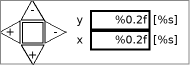
VISUALIZATION _VISU_PlacementXY_cross  // 190x65
VAR_IN_OUT
	m_Inst : FB_PointCorr;  
END_VAR
    Polyline (21,20) (32,0) (44,20) (21,20), "-"
        p3092690914: m_Inst.nBtnColor
        tap m_Inst.bCmd_Y_minus
    Polyline (21,45) (33,65) (44,45) (21,45), "+"
        p3092690914: m_Inst.nBtnColor
        tap m_Inst.bCmd_Y_plus
    Polyline (45,43) (45,21) (66,32) (45,43), "-"
        p3092690914: m_Inst.nBtnColor
        tap m_Inst.bCmd_X_minus
    Polyline (20,43) (20,21) (0,32) (20,43), "+"
        p3092690914: m_Inst.nBtnColor
        tap m_Inst.bCmd_X_plus
    Rectangle (70,30 20x20), "x"
    Rectangle (70,10 20x20), "y"
    Rectangle (22,22 21x21)
    Rectangle (150,10 40x20), "[%s]", text variable: m_Inst._aUnit
    Rectangle (150,30 40x20), "[%s]", text variable: m_Inst._aUnit
    Rectangle (90,10 60x20), "%0.2f", text variable: m_Inst.fY_Pos
        OnMouseClick: write the text variable via Default
    Rectangle (90,30 60x20), "%0.2f", text variable: m_Inst.fX_Pos
        OnMouseClick: write the text variable via Default
END_VISUALIZATION

(* stored: Version 1.1.0.1, ProductVersion 3.1.4024.3
   Visu _VISU_PlacementXY_cross: Id {4b279807-5098-448c-81d2-932d3c8860ad} *)
